// TIA Portal V16 export
// export: Created 2021-04-06T19:52:16.6360998Z, ExportSetting WithDefaults, DisplayName Totally Integrated Automation Portal, DisplayVersion V16, DisplayName TIA Portal Version Control Interface, DisplayVersion V16, DisplayName TIA Portal Openness, DisplayVersion V16, DisplayName STEP 7 Professional, DisplayVersion V16, DisplayName STEP 7 Safety, DisplayVersion V16, DisplayName WinCC Unified SCADA Engineering System, DisplayVersion V16
FUNCTION_BLOCK "workVibroLot_AM"   // FB8, LAD
TITLE = Управление линиями вибролотков и вибраций
{ S7_Optimized_Access := 'TRUE' }
VERSION : 0.1
// Если собрано разрешение на работу и ReadyToSort=0 и если вес меньше заданного то включен вибролоток и открыта лопатка
// stored: AutoNumber true, IsIECCheckEnabled false, IsRetainMemResEnabled false, MemoryReserve 100, SetENOAutomatically false, UDAEnableTagReadback false
   VAR_INPUT
      enableWork : Bool;   // разрешение работы
      setWeightBunker : Real;   // уставка веса для бункера
      currentWeight : Real;   // текущий вес
      stateDoor : Bool;   // состояние лопатки
      stateBunkerLeft : Bool;   // состояние левого бункера
      stateBunkerRight : Bool;   // состояние правого бункера
      isWorkWithBunker : Bool;   // разрешение работать с конкретными бункерами
   END_VAR
   VAR_IN_OUT
      onVibroLot : Bool;   // сигнал на включение вибролотков
      closeDoor : Bool;   // сигнал на закрытие лопатки
      openDoor : Bool;   // сигнал на открытие лопатки
      alarmStop : Bool;   // аварийный останов
      isReadyToSort : Bool;   // бункер готов к сортировке
      isReadyToDrop : Bool;   // бункер готов к сбросу
   END_VAR
   VAR
      controlDoor : "controlValve";
      enableWorkAfterCloseDoor : Bool;   // разрешение работы после закрытия бункеров
      tonAfterCloseDoor : TON_TIME;   // выдержка времени после закрытия бункеров
      stateBothBunker : Bool;   // состояние обоих бункеров
      tonToSetSort : TON_TIME;   // выдержка на выставление готов к сортировке
      startToToSetSort : Bool;   // бит на старт таймера выше
      isSetSort : Bool;   // сигнал что бункер готов к сортировке
   END_VAR
   VAR_TEMP
      tmpOpen : Bool;
      tmpClose : Bool;
   END_VAR
BEGIN

REGION Network 1 (SCL): состояние обоих бункеров
   //определим состояние бункеров
   #stateBothBunker := NOT (#stateBunkerLeft) AND NOT (#stateBunkerRight);

   //сигнал выдержки на разрешение работы лотка
   #tonAfterCloseDoor(IN:=#stateBothBunker,
                      PT:=t#300ms,
                      Q=>#enableWorkAfterCloseDoor);
   //сигнал выдержки для выставления состояния готов к сортировке
   #tonToSetSort(IN := #startToToSetSort,
                 PT := t#250ms,
                 Q => #isSetSort);

   IF #isSetSort THEN
       #isReadyToSort := true;
       #startToToSetSort := false;
   END_IF;

   IF #enableWork AND NOT(#alarmStop) THEN//проверяем глобальное разрешение на работу
       IF #currentWeight < #setWeightBunker THEN
           #isReadyToSort := false;
       END_IF;
       IF  #currentWeight<#setWeightBunker AND NOT(#isReadyToSort)
           AND NOT(#isReadyToDrop) AND #isWorkWithBunker
           AND #enableWorkAfterCloseDoor
       THEN
           #startToToSetSort := FALSE;
           #onVibroLot := true;
           IF NOT (#stateDoor) THEN
               #tmpOpen := true;
           END_IF;

       ELSE
           //если мы зашли сюда потому что набрали вес, то заупускаем таймер
           IF #currentWeight >= #setWeightBunker AND NOT(#isReadyToDrop)
               AND NOT(#isReadyToSort) AND #enableWorkAfterCloseDoor THEN
               #startToToSetSort := true;
           END_IF;
           //если зашли сюда потому что уже таймер вышел либо, готовы к сбросу,
           //либо нет разрешений то просто держим лоток выключенным и закрытым
           IF #isReadyToDrop OR #isReadyToSort
               OR NOT(#enableWorkAfterCloseDoor) OR NOT(#isWorkWithBunker)  THEN
               #onVibroLot := false;
               IF #stateDoor THEN
                   #tmpClose := true;
               END_IF;
           END_IF;


       END_IF;

   ELSE
       #isSetSort := false;
       #startToToSetSort := false;
       #isReadyToSort := FALSE;
       #onVibroLot := FALSE;
       #openDoor := FALSE;
       #closeDoor := false;
   END_IF;





   //управление лопаткой
   #controlDoor("time_open/close" := T#250ms,
                openQ => #openDoor,
                closeQ => #closeDoor,
                open := #tmpOpen,
                close := #tmpClose,
                stopAlarm := #alarmStop);
END_REGION
END_FUNCTION_BLOCK
